TYPE "TMeasuring_ERRORWORD"
VERSION : 0.1
// Block: TMeasuring_ERRORWORD
   STRUCT
      SystemFault : Bool;
      ConfigFault : Bool;
      UserFault : Bool;
      CommandNotAccepted : Bool;
      PeripheralError : Bool;
   END_STRUCT;

END_TYPE
